Staubli VAL3: start.pgx

program start()
begin
  call Deb2304()
end
